# EPICS autosave request: ESP300/iocBoot/ioc_esp_bmc/auto_settings.req
file "XFM_motor_settings.req",        P=XF:04BMC-ES:, M=DET:1-Ax:Y:Mtr
